TYPE STR :
STRUCT
		MesIdc			: REAL;   						(* (A) DC current *)
		MesUdc			: REAL;							(* (V) DC voltage *)
END_STRUCT
END_TYPE

(* stored: Version 1.1.0.1, ProductVersion 3.1.4024.9
   DUT STR: Id {0d4fde0f-a3da-451f-85d8-d101d296b309} *)
